FUNCTION_BLOCK ROBOT_DATA_HANDLER
VAR_INPUT
END_VAR
VAR_OUTPUT
END_VAR
VAR
END_VAR

METHOD PUBLIC DATA_TO_STRING : STRING
VAR_INPUT
END_VAR
VAR
	emptyJointsString : STRING := '0.0 0.0 0.0 0.0 0.0';
	separator : STRING := ' ';
	
	debugValue : LREAL := 10.0;
END_VAR
// CONVERT MOVEMENT DATA TO ROBOT MOVEMENT STRING.

//GVL.robotData.joint0.speed := 0.0; // DEBUG REMOVE LATER
//GVL.robotData.joint1.speed := 0.0; // DEBUG REMOVE LATER
//GVL.robotData.joint2.speed := 0.0; // DEBUG REMOVE LATER
//GVL.robotData.joint3.speed := 0.0; // DEBUG REMOVE LATER

DATA_TO_STRING :=
	CONCAT(LREAL_TO_STRING(GVL.robotData.joint0.curSpeed), 
	CONCAT(separator, 
	CONCAT(LREAL_TO_STRING(GVL.robotData.joint1.curSpeed),
	CONCAT(separator, 
	CONCAT(LREAL_TO_STRING(GVL.robotData.joint2.curSpeed),
	CONCAT(separator,  
	CONCAT(LREAL_TO_STRING(GVL.robotData.joint3.curSpeed),
	CONCAT(separator,
		emptyJointsString))))))));
END_METHOD

METHOD PUBLIC DEGREES_TO_MOVEMENT_DATA : BOOL
VAR_INPUT
	degrees : LREAL;
	jointNr : INT;
END_VAR
VAR
	moveTime : TIME;
	moveSpeed : LREAL;
	tempTimeValue : LREAL;
	speedMultiplier : LREAL := 3;
	TimePerDegree : LREAL := 544;
	TimePerDegree3 : LREAL := 390;
	tempDegrees : LREAL;
END_VAR
CASE jointNr OF
	0:
		tempDegrees := degrees - GVL.robotData.joint0.curPosition;
	1:
		tempDegrees := degrees - GVL.robotData.joint1.curPosition;
	2:
		tempDegrees := degrees - GVL.robotData.joint2.curPosition;
	3:
		tempDegrees := degrees - GVL.robotData.joint3.curPosition;
END_CASE

IF (tempDegrees < 0) THEN
	moveSpeed := 20.0;
	tempDegrees := tempDegrees * -1;
ELSIF (tempDegrees > 0) THEN
	moveSpeed := -20.0;
	tempDegrees := tempDegrees;
END_IF


moveSpeed := moveSpeed * speedMultiplier;
IF (jointNr = 3) THEN
	tempTimeValue := ((tempDegrees * TimePerDegree3) / speedMultiplier);
ELSE
	tempTimeValue := ((tempDegrees * TimePerDegree) / speedMultiplier);
END_IF
moveTime := LREAL_TO_TIME(tempTimeValue);


CASE jointNr OF
	0:
		GVL.robotData.joint0.timer.timerTime := moveTime;
		GVL.robotData.joint0.setSpeed := moveSpeed;
		GVL.robotData.joint0.curPosition := degrees;
	1:
		GVL.robotData.joint1.timer.timerTime := moveTime;
		GVL.robotData.joint1.setSpeed := moveSpeed;
		GVL.robotData.joint1.curPosition := degrees;
	2:
		GVL.robotData.joint2.timer.timerTime := moveTime;
		GVL.robotData.joint2.setSpeed := moveSpeed;
		GVL.robotData.joint2.curPosition := degrees;
	3:
		GVL.robotData.joint3.timer.timerTime := moveTime;
		GVL.robotData.joint3.setSpeed := moveSpeed;
		GVL.robotData.joint3.curPosition := degrees;
END_CASE
END_METHOD

METHOD PUBLIC JOINT_DATA_HANDLER : BOOL
VAR_INPUT
END_VAR
// TURN RECEIVED ROBOT DATA INTO CURRENT JOINTS POSITIONS
// DONT USE THIS METHOD!!!!!!!!!!

IF (GVL.ReceivedStringArray[0] = 'CRISTART') THEN
	// WHAT IS THE LOCATION
END_IF


// WE CAN'T GET THE CURRENT LOCATION FROM THE ROBOT SO WE LEFT THIS EMPTY FOR NOW!!
END_METHOD

METHOD PUBLIC MOVEMENT_CONTROLLER : BOOL
VAR_INPUT
END_VAR
VAR
	count : INT := 0;
END_VAR
FOR count := 0 TO 3 BY 1 DO
	CASE count OF
		0:
			IF (GVL.robotData.joint0.setSpeed <> 0 AND GVL.robotData.isBusy[4] = FALSE) THEN
				GVL.robotData.joint0.timer.timerStart := TRUE;
				GVL.robotData.joint0.curSpeed := GVL.robotData.joint0.setSpeed;
				GVL.robotData.joint0.setSpeed := 0;
				GVL.robotData.isBusy[0] := TRUE;
			ELSIF(GVL.robotData.joint0.timer.timerCon.Q) THEN
				GVL.robotData.joint0.timer.timerStart := FALSE;
				GVL.robotData.joint0.curSpeed := 0.0;
				GVL.robotData.isBusy[0] := FALSE;
			END_IF
		1:
			IF (GVL.robotData.joint1.setSpeed <> 0 AND GVL.robotData.isBusy[4] = FALSE) THEN
				GVL.robotData.joint1.timer.timerStart := TRUE;
				GVL.robotData.joint1.curSpeed := GVL.robotData.joint1.setSpeed;
				GVL.robotData.joint1.setSpeed := 0;
				GVL.robotData.isBusy[1] := TRUE;
			ELSIF(GVL.robotData.joint1.timer.timerCon.Q) THEN
				GVL.robotData.joint1.timer.timerStart := FALSE;
				GVL.robotData.joint1.curSpeed := 0.0;
				GVL.robotData.isBusy[1] := FALSE;
			END_IF
		2:
			IF (GVL.robotData.joint2.setSpeed <> 0 AND GVL.robotData.isBusy[4] = FALSE) THEN
				GVL.robotData.joint2.timer.timerStart := TRUE;
				GVL.robotData.joint2.curSpeed := GVL.robotData.joint2.setSpeed;
				GVL.robotData.joint2.setSpeed := 0;
				GVL.robotData.isBusy[2] := TRUE;
			ELSIF(GVL.robotData.joint2.timer.timerCon.Q) THEN
				GVL.robotData.joint2.timer.timerStart := FALSE;
				GVL.robotData.joint2.curSpeed := 0.0;
				GVL.robotData.isBusy[2] := FALSE;
			END_IF
		3:
			IF (GVL.robotData.joint3.setSpeed <> 0 AND GVL.robotData.isBusy[4] = FALSE) THEN
				GVL.robotData.joint3.timer.timerStart := TRUE;
				GVL.robotData.joint3.curSpeed := GVL.robotData.joint3.setSpeed;
				GVL.robotData.joint3.setSpeed := 0;
				GVL.robotData.isBusy[3] := TRUE;
			ELSIF(GVL.robotData.joint3.timer.timerCon.Q) THEN
				GVL.robotData.joint3.timer.timerStart := FALSE;
				GVL.robotData.joint3.curSpeed := 0.0;
				GVL.robotData.isBusy[3] := FALSE;
			END_IF
	END_CASE
END_FOR

IF (GVL.robotData.isBusy[0] = FALSE AND GVL.robotData.isBusy[1] = FALSE AND GVL.robotData.isBusy[2] = FALSE AND GVL.robotData.isBusy[3] = FALSE) THEN
	GVL.robotData.isBusy[4] := FALSE;
ELSE
	GVL.robotData.isBusy[4] := TRUE;
END_IF
END_METHOD

METHOD PUBLIC TARGET_TO_DEGREES_CALCULATOR : BOOL
VAR_INPUT
END_VAR
// TURN CURRENT POSITION AND TARGET POSITION TO INTO MOVEMENT PER JOINT.
END_METHOD

END_FUNCTION_BLOCK

(* stored: Version 1.1.0.1, ProductVersion 3.1.4024.12
   POU ROBOT_DATA_HANDLER: Id {e0987821-00dd-4921-8e97-ded148e1ea82}, SpecialFunc None
   Method DATA_TO_STRING: Id {fccde642-b27d-4984-8d27-e867d0497562}
   Method DEGREES_TO_MOVEMENT_DATA: Id {0af9d1a1-3d38-4078-9a1c-ac12d9d574c7}
   Method JOINT_DATA_HANDLER: Id {950a9264-99be-412c-ae5a-e97f094a88ef}
   Method MOVEMENT_CONTROLLER: Id {6693a925-8cf1-4973-8966-fef29abe4757}
   Method TARGET_TO_DEGREES_CALCULATOR: Id {75f14b1b-a7a8-462d-a304-4bcbb1ec7ecf} *)
